// TIA Portal V21 export
TYPE "lubricationSystemConfig"
   STRUCT
      almMask : DWord := 16#FFFFFFFF;
      timeToEstablishReturnFlow : Time := T#15s;
      noFlowDelay : Time := T#5s;
      maxStopTime : Time := T#5s;
      oilTempHeaterSp : Real := 32.5;
      oilTempHeaterHyst : Real := 2.5;
      oilTempCoolerSp : Real := 41.5;
      oilTempCoolerHyst : Real := 1.5;
      timeToEstablishFlow : Time := T#5s;
      minOilFlow : Real := 165.0;   // l/m
   END_STRUCT;
END_TYPE
